(* Logix 5000 project; controller HP_SSC01hv vendor 1 type 14 code 158 rev 32.11; software revision 32.03; part 5 of 15 *)
(* tags used below, declared in another part *)
   A_C2_0300 : ALIAS FOR C2_FaultStandard.0;
   A_C2_0301 : ALIAS FOR C2_FaultStandard.1;
   A_C2_0302 : ALIAS FOR C2_FaultStandard.2;
   A_C2_0303 : ALIAS FOR C2_FaultStandard.3;
   A_C2_0305 : ALIAS FOR C2_FaultStandard.5;
   A_C2_0309 : ALIAS FOR C2_FaultStandard.9;
   A_C2_0310 : ALIAS FOR C2_FaultStandard.10;
   A_C2_0311 : ALIAS FOR C2_FaultStandard.11;
   A_C2_0312 : ALIAS FOR C2_FaultStandard.12;
   A_C2_0313 : ALIAS FOR C2_FaultStandard.13;
   A_C2_0314 : ALIAS FOR C2_FaultStandard.14;
   A_C2_0315 : ALIAS FOR C2_FaultStandard.15;
   A_C2_0317 : ALIAS FOR C2_FaultStandard.17;
   A_C2_0319 : ALIAS FOR C2_FaultStandard.19;
   A_C2_0321 : ALIAS FOR C2_FaultStandard.21;
   A_C2_0322 : ALIAS FOR C2_FaultStandard.22;
   A_C2_0323 : ALIAS FOR C2_FaultStandard.23;
   A_C2_0324 : ALIAS FOR C2_FaultStandard.24;
   A_C2_0325 : ALIAS FOR C2_FaultStandard.25;
   A_C2_0327 : ALIAS FOR C2_FaultStandard.27;
   A_C2_0328 : ALIAS FOR C2_FaultStandard.28;
   A_C2_0329 : ALIAS FOR C2_FaultStandard.29;
   A_C2_0330 : ALIAS FOR C2_FaultStandard.30;
   A_C2_0331 : ALIAS FOR C2_FaultStandard.31;
   A_C2_0404 : ALIAS FOR C2_Warning.4;
   A_C2_0406 : ALIAS FOR C2_Warning.6;
   A_C2_0407 : ALIAS FOR C2_Warning.7;
   A_C2_0408 : ALIAS FOR C2_Warning.8;
   A_C2_0409 : ALIAS FOR C2_Warning.9;
   A_C2_0412 : ALIAS FOR C2_Warning.12;
   A_C2_0413 : ALIAS FOR C2_Warning.13;
   A_C2_0414 : ALIAS FOR C2_Warning.14;
   A_C2_0415 : ALIAS FOR C2_Warning.15;
   A_C2_0416 : ALIAS FOR C2_Warning.16;
   A_C2_0424 : ALIAS FOR C2_Warning.24;
   A_C2_0427 : ALIAS FOR C2_Warning.27;
   A_C2_0428 : ALIAS FOR C2_Warning.28;
   A_C2_0430 : ALIAS FOR C2_Warning.30;
   C2_32HourTimers : TIMER[4];
   C2_All_DLY_OK : BOOL;
   C2_BrakeSequenceInProcess : BOOL;
   C2_BrakeTest : BOOL;
   C2_BrakeTestEndPosition : REAL;
   C2_BrakeTestFailed : BOOL;
   C2_BrakeTestLocalDisable : BOOL;
   C2_BrakeTestMAJ01 : MOTION_INSTRUCTION;
   C2_BrakeTestMessageNumber : DINT;
   C2_BrakeTestONS : BOOL;
   C2_BrakeTestSelected : BOOL;
   C2_BrakeTestSequence : DINT;
   C2_BrakeTestSequenceAlarms : DINT;
   C2_BrakeTestSequenceAlarmTimer : TIMER[16];
   C2_BrakeTestSequenceONS : DINT;
   C2_BrakeTestStartPosition : REAL;
   C2_BrakeTestStoppingDistance : REAL;
   C2_BrakeTestTimerHoldVel : TIMER;
   C2_BrakeTestWarning : BOOL;
   C2_DisableTimer : TIMER;
   C2_DumpTest : BOOL;
   C2_DumpValveFailedOff : BOOL;
   C2_DumpValveFailedOn : BOOL;
   C2_DumpValveMessageNumber : DINT;
   C2_DumpValveTestDelay : TIMER[4];
   C2_DumpValveTestDelay2 : TIMER;
   C2_DumpValveTestSelected : BOOL;
   C2_DumpValveTestSequence : DINT;
   C2_DumpValveTestSequenceAlarms : DINT;
   C2_DumpValveTestSequenceAlarmTimer : TIMER[8];
   C2_EncoderCounts : DINT;
   C2_EncoderCountsRaw : ALIAS FOR C2_RIO_AENT:3:I.PresentData;
   C2_EncoderDegree : REAL;
   C2_FaultDebounce : TIMER[16];
   C2_FaultHoldTimer : TIMER[4];
   C2_FaultHomeSwitchNotFound : BOOL;
   C2_FaultStandard : DINT;
   C2_HomeInputStatus : BOOL;
   C2_HomeSequence : DINT;
   C2_HomeSequenceAlarms : DINT;
   C2_HomeSwitchFaultK7KFailedOff : BOOL;
   C2_HomeSwitchFaultK7KFailedOn : BOOL;
   C2_HomeSwitchFaultSafeFailedOff : BOOL;
   C2_HomeSwitchFaultSafeFailedOn : BOOL;
   C2_IndexEnable : BOOL;
   C2_JogEnable : BOOL;
   C2_LIM_ALARM_B : ALIAS FOR C2_RIO_AENT:I.Data[1].0;
   C2_MaintEnable : BOOL;
   C2_MotorActualPositionX1000 : DINT;
   C2_MotorAverageVelocityX1000 : DINT;
   C2_MotorFan : ALIAS FOR C2_RIO_AENT:O.Data[2].0;
   C2_MSF : MOTION_INSTRUCTION;
   C2_MSO : MOTION_INSTRUCTION;
   C2_OIT_Current : DINT;
   C2_ONS_Fault : DINT;
   C2_RemoteBrakeAndHomeSequenceAlarms : DINT;
   C2_RemoteBrakeTestCMD : BOOL;
   C2_RemoteDumpTestCMD : BOOL;
   C2_ServoActionStatusOffDelay : TIMER;
   C2_ServoActionStatusOnDelay : TIMER;
   C2_ServoFanOverload : ALIAS FOR C2_RIO_AENT:I.Data[1].2;
   C2_SS_LocalRemote_1_IsRemote : ALIAS FOR C2_RIO_AENT:I.Data[1].3;
   C2_SS_RemoteMode : BOOL;
   C2_Warning : DINT;
   C2DumpValveTestSequenceONS : DINT;
   none : BOOL;
   RCS_CMD_RunInAuto : BOOL;
   RCS_SyncMotionEnable : BOOL;
   S_C2_EncoderPositionDegree : DINT;
   S_C2_ExecutePB : BOOL;
   S_C2_FaultReset : BOOL;
   S_C2_ModeLocal : BOOL;
   S_C2_ModeRemote : BOOL;
   S_C2_MotionEnabled : BOOL;
   S_C2_MSTOP_InputOK : BOOL;
   S_C2_NearOnPath : BOOL;
   S_C2_OffPath : BOOL;
   S_C2_OIT_FaultReset : BOOL;
   S_C2_OutputEnable : BOOL;
   S_C2_PressureOK : ALIAS FOR C2_Safe:I.Pt05Data;
   S_C2_SAFETY_ENABLE_1 : ALIAS FOR C2_Safe:O.Pt00Data;
   S_C2_SAFETY_ENABLE_2 : ALIAS FOR C2_Safe:O.Pt01Data;
   S_C2_Stop1_OK : BOOL;
   S_RCS_CMD_FaultReset : BOOL;
   STS_Enable_Rail : DINT;
   ZZZ_DIAG_A_C2_0302 : BOOL;
   ZZZ_DIAG_C2_AxisFault : DINT;
   ZZZ_DIAG_C2_AxisStatus : DINT;
   ZZZ_DIAG_C2_EnableRail : DINT;
   ZZZ_DIAG_C2_MotionStatus : DINT;
   ZZZ_DIAG_C2_MSF : MOTION_INSTRUCTION;
   ZZZ_DIAG_C2_MSO : MOTION_INSTRUCTION;
   ZZZ_DIAG_C2_OneTimeOnly : BOOL;
   ZZZ_DIAG_C2_OutputEnable : BOOL;
   ZZZ_DIAG_C2_OutputEnable_ACC : DINT;
   ZZZ_DIAG_ONS : DINT;
   ZZZ_DIAG_S_C2_OutputEnableTON : TIMER;
   ZZZ_DIAG_S_C2_SAFETY_ENABLE_1 : BOOL;
   ZZZ_DIAG_S_C2_SAFETY_ENABLE_2 : BOOL;

PROGRAM Carousel2   (* main routine C200_Main *)
VAR
   zzz_Test20 : BOOL;
   zzz_Test21 : BOOL;
END_VAR

ROUTINE C200_Main   (* ladder *)
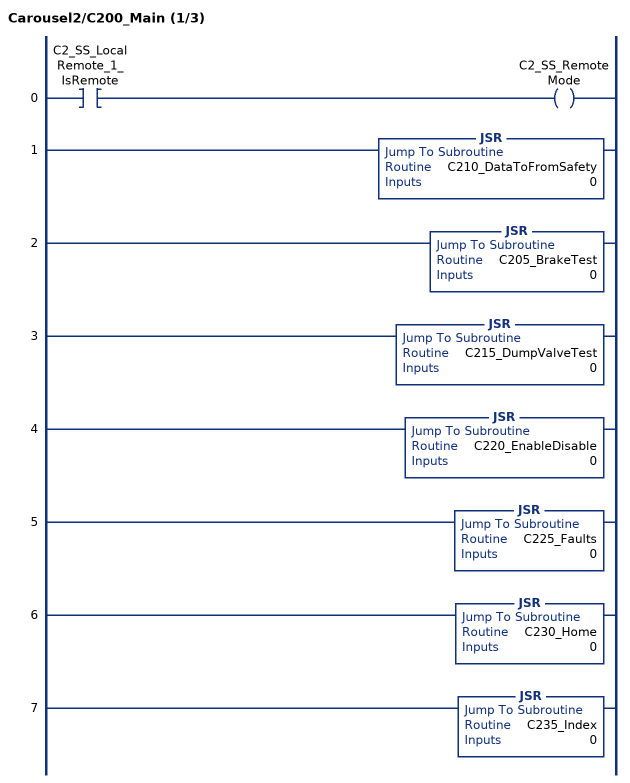
   0: XIC(C2_SS_LocalRemote_1_IsRemote)OTE(C2_SS_RemoteMode);
   1: JSR(C210_DataToFromSafety,0);
   2: JSR(C205_BrakeTest,0);
   3: JSR(C215_DumpValveTest,0);
   4: JSR(C220_EnableDisable,0);
   5: JSR(C225_Faults,0);
   6: JSR(C230_Home,0);
   7: JSR(C235_Index,0);
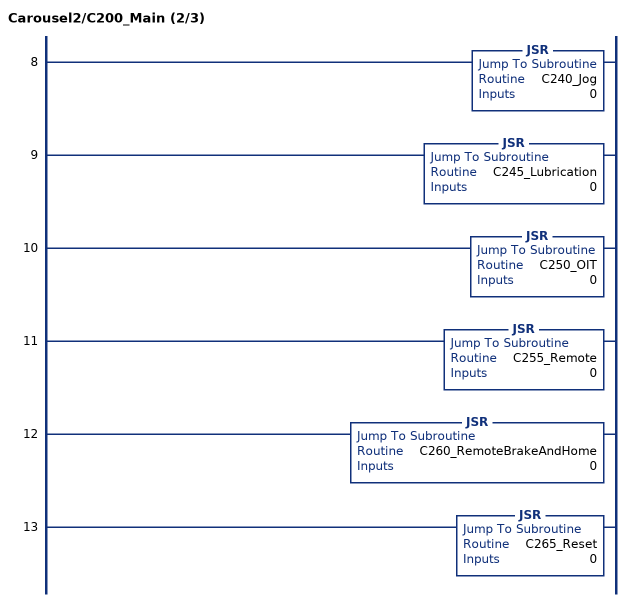
   8: JSR(C240_Jog,0);
   9: JSR(C245_Lubrication,0);
   10: JSR(C250_OIT,0);
   11: JSR(C255_Remote,0);
   12: JSR(C260_RemoteBrakeAndHome,0);
   13: JSR(C265_Reset,0);
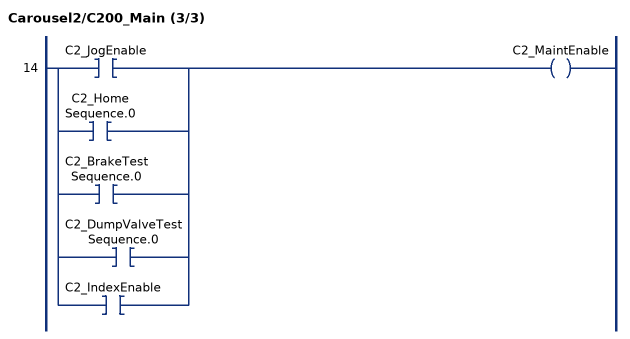
   14: [XIC(C2_JogEnable) ,XIC(C2_HomeSequence.0) ,XIC(C2_BrakeTestSequence.0) ,XIC(C2_DumpValveTestSequence.0) ,XIC(C2_IndexEnable) ]OTE(C2_MaintEnable);
END_ROUTINE

ROUTINE C205_BrakeTest   (* ladder *)
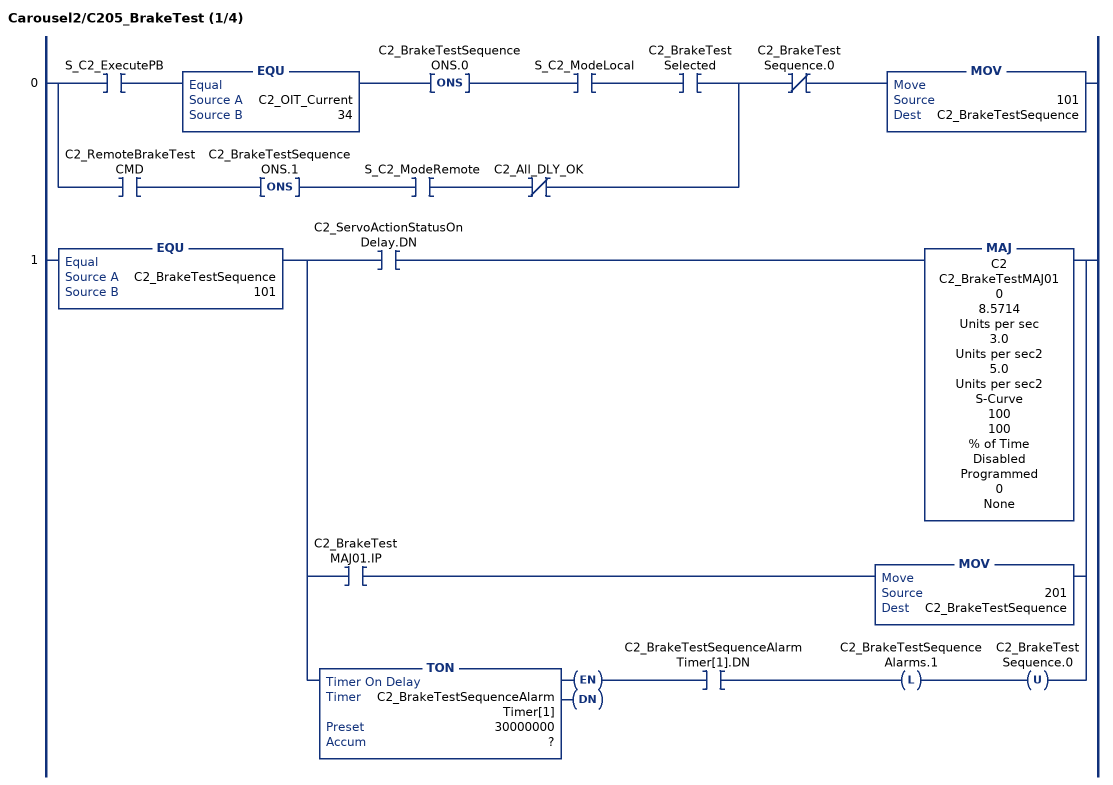
   0: [XIC(S_C2_ExecutePB) EQU(C2_OIT_Current,34) ONS(C2_BrakeTestSequenceONS.0) XIC(S_C2_ModeLocal) XIC(C2_BrakeTestSelected) ,XIC(C2_RemoteBrakeTestCMD) ONS(C2_BrakeTestSequenceONS.1) XIC(S_C2_ModeRemote) XIO(C2_All_DLY_OK) ]XIO(C2_BrakeTestSequence.0)MOV(101,C2_BrakeTestSequence);
   1: EQU(C2_BrakeTestSequence,101)[XIC(C2_ServoActionStatusOnDelay.DN) MAJ(C2,C2_BrakeTestMAJ01,0,8.5714,Units per sec,3.0,Units per sec2,5.0,Units per sec2,S-Curve,100,100,% of Time,Disabled,Programmed,0,None) ,XIC(C2_BrakeTestMAJ01.IP) MOV(201,C2_BrakeTestSequence) ,TON(C2_BrakeTestSequenceAlarmTimer[1],?,?) XIC(C2_BrakeTestSequenceAlarmTimer[1].DN) OTL(C2_BrakeTestSequenceAlarms.1) OTU(C2_BrakeTestSequence.0) ];
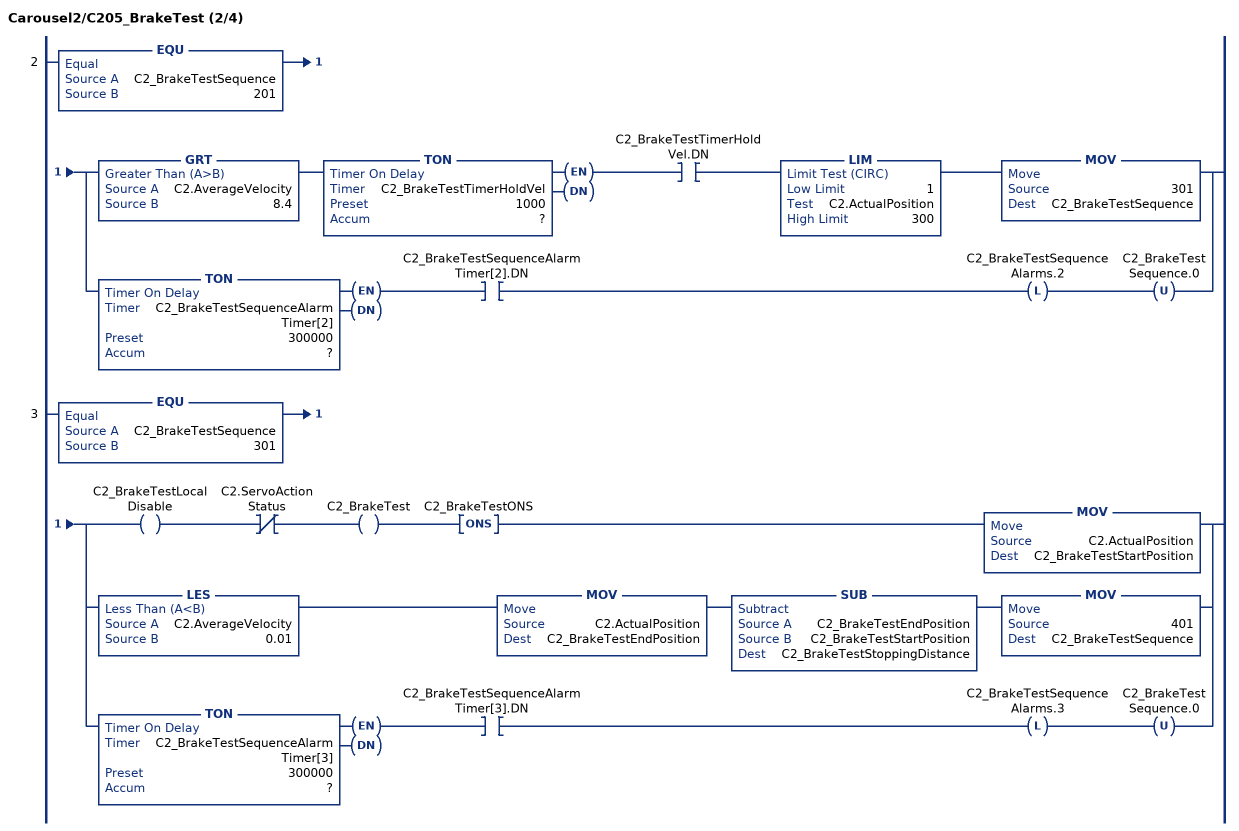
   2: EQU(C2_BrakeTestSequence,201)[GRT(C2.AverageVelocity,8.4) TON(C2_BrakeTestTimerHoldVel,?,?) XIC(C2_BrakeTestTimerHoldVel.DN) LIM(1,C2.ActualPosition,300) MOV(301,C2_BrakeTestSequence) ,TON(C2_BrakeTestSequenceAlarmTimer[2],?,?) XIC(C2_BrakeTestSequenceAlarmTimer[2].DN) OTL(C2_BrakeTestSequenceAlarms.2) OTU(C2_BrakeTestSequence.0) ];
   3: EQU(C2_BrakeTestSequence,301)[OTE(C2_BrakeTestLocalDisable) XIO(C2.ServoActionStatus) OTE(C2_BrakeTest) ONS(C2_BrakeTestONS) MOV(C2.ActualPosition,C2_BrakeTestStartPosition) ,LES(C2.AverageVelocity,0.01) MOV(C2.ActualPosition,C2_BrakeTestEndPosition) SUB(C2_BrakeTestEndPosition,C2_BrakeTestStartPosition,C2_BrakeTestStoppingDistance) MOV(401,C2_BrakeTestSequence) ,TON(C2_BrakeTestSequenceAlarmTimer[3],?,?) XIC(C2_BrakeTestSequenceAlarmTimer[3].DN) OTL(C2_BrakeTestSequenceAlarms.3) OTU(C2_BrakeTestSequence.0) ];
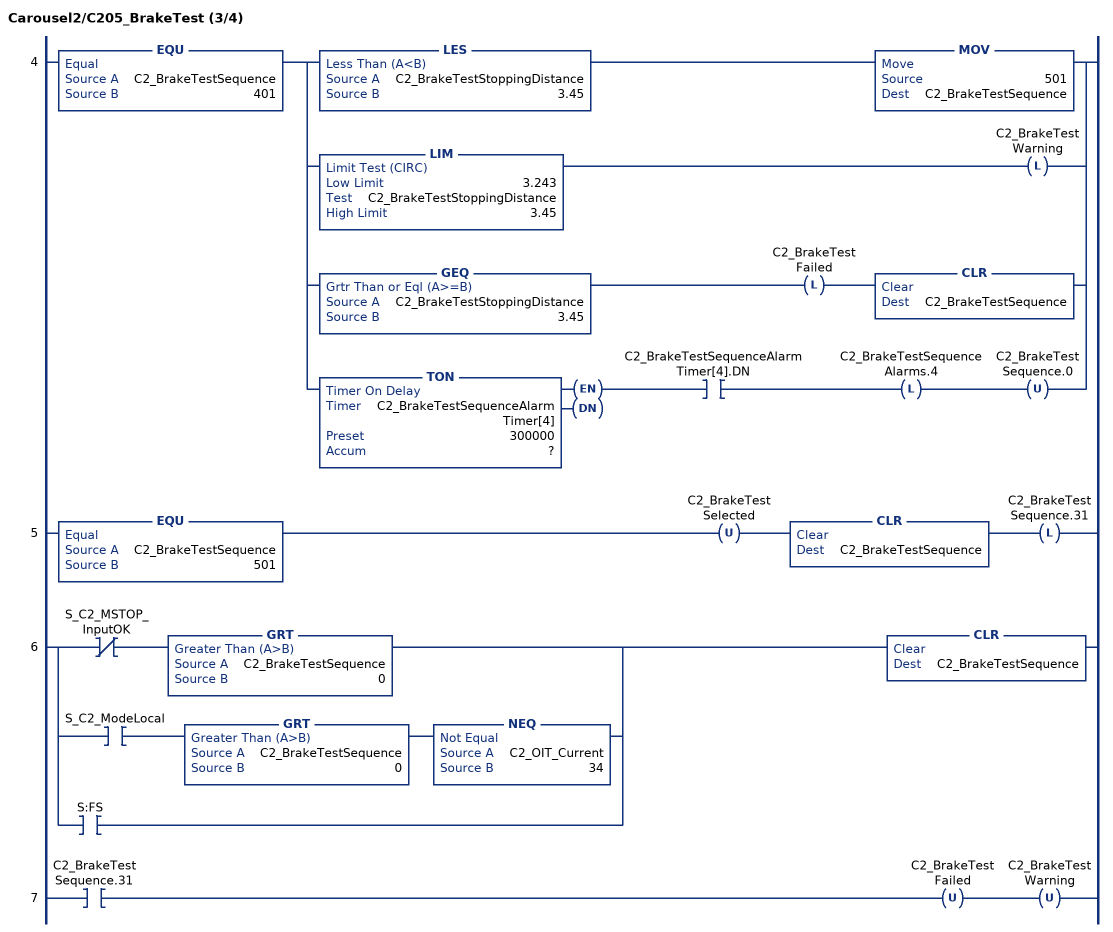
   4: EQU(C2_BrakeTestSequence,401)[LES(C2_BrakeTestStoppingDistance,3.45) MOV(501,C2_BrakeTestSequence) ,LIM(3.243,C2_BrakeTestStoppingDistance,3.45) OTL(C2_BrakeTestWarning) ,GEQ(C2_BrakeTestStoppingDistance,3.45) OTL(C2_BrakeTestFailed) CLR(C2_BrakeTestSequence) ,TON(C2_BrakeTestSequenceAlarmTimer[4],?,?) XIC(C2_BrakeTestSequenceAlarmTimer[4].DN) OTL(C2_BrakeTestSequenceAlarms.4) OTU(C2_BrakeTestSequence.0) ];
   5: EQU(C2_BrakeTestSequence,501)OTU(C2_BrakeTestSelected)CLR(C2_BrakeTestSequence)OTL(C2_BrakeTestSequence.31);
   6: [XIO(S_C2_MSTOP_InputOK) GRT(C2_BrakeTestSequence,0) ,XIC(S_C2_ModeLocal) GRT(C2_BrakeTestSequence,0) NEQ(C2_OIT_Current,34) ,XIC(S:FS) ]CLR(C2_BrakeTestSequence);
   7: XIC(C2_BrakeTestSequence.31)OTU(C2_BrakeTestFailed)OTU(C2_BrakeTestWarning);
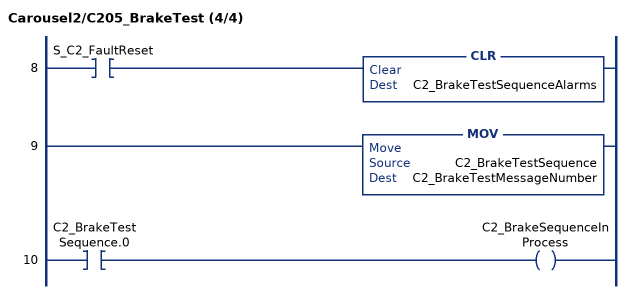
   8: XIC(S_C2_FaultReset)CLR(C2_BrakeTestSequenceAlarms);
   9: MOV(C2_BrakeTestSequence,C2_BrakeTestMessageNumber);
   10: XIC(C2_BrakeTestSequence.0)OTE(C2_BrakeSequenceInProcess);
END_ROUTINE

ROUTINE C210_DataToFromSafety   (* ladder *)
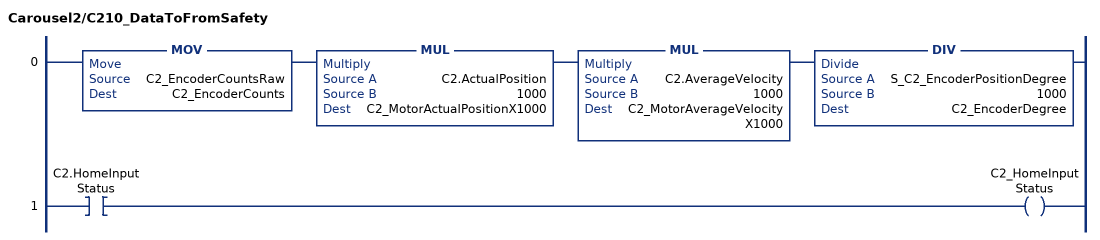
   0: MOV(C2_EncoderCountsRaw,C2_EncoderCounts)MUL(C2.ActualPosition,1000,C2_MotorActualPositionX1000)MUL(C2.AverageVelocity,1000,C2_MotorAverageVelocityX1000)DIV(S_C2_EncoderPositionDegree,1000,C2_EncoderDegree);
   1: XIC(C2.HomeInputStatus)OTE(C2_HomeInputStatus);
END_ROUTINE

ROUTINE C215_DumpValveTest   (* ladder *)
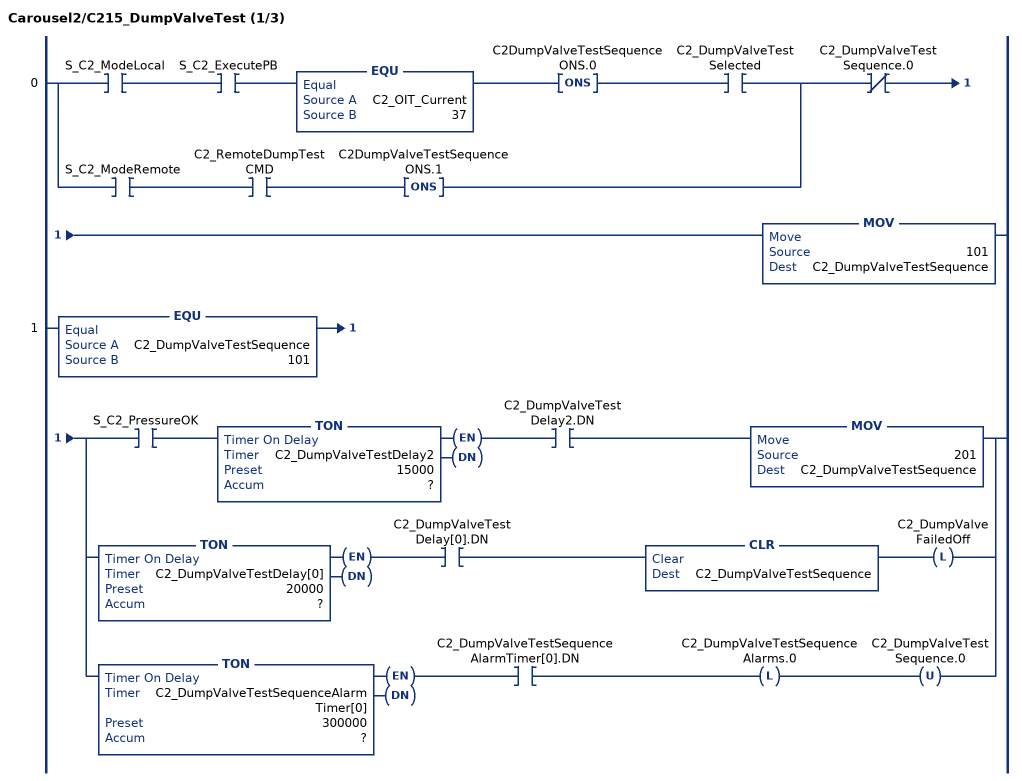
   0: [XIC(S_C2_ModeLocal) XIC(S_C2_ExecutePB) EQU(C2_OIT_Current,37) ONS(C2DumpValveTestSequenceONS.0) XIC(C2_DumpValveTestSelected) ,XIC(S_C2_ModeRemote) XIC(C2_RemoteDumpTestCMD) ONS(C2DumpValveTestSequenceONS.1) ]XIO(C2_DumpValveTestSequence.0)MOV(101,C2_DumpValveTestSequence);
   1: EQU(C2_DumpValveTestSequence,101)[XIC(S_C2_PressureOK) TON(C2_DumpValveTestDelay2,?,?) XIC(C2_DumpValveTestDelay2.DN) MOV(201,C2_DumpValveTestSequence) ,TON(C2_DumpValveTestDelay[0],?,?) XIC(C2_DumpValveTestDelay[0].DN) CLR(C2_DumpValveTestSequence) OTL(C2_DumpValveFailedOff) ,TON(C2_DumpValveTestSequenceAlarmTimer[0],?,?) XIC(C2_DumpValveTestSequenceAlarmTimer[0].DN) OTL(C2_DumpValveTestSequenceAlarms.0) OTU(C2_DumpValveTestSequence.0) ];
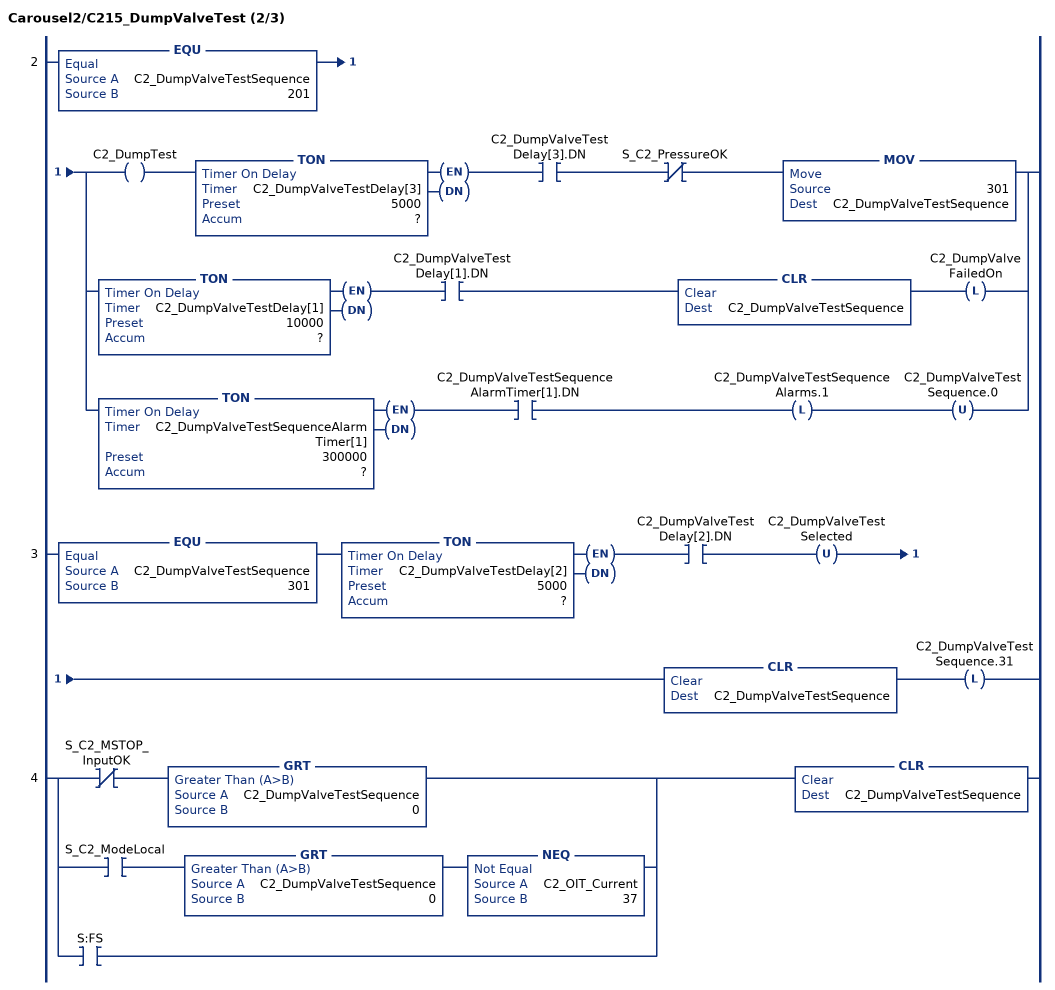
   2: EQU(C2_DumpValveTestSequence,201)[OTE(C2_DumpTest) TON(C2_DumpValveTestDelay[3],?,?) XIC(C2_DumpValveTestDelay[3].DN) XIO(S_C2_PressureOK) MOV(301,C2_DumpValveTestSequence) ,TON(C2_DumpValveTestDelay[1],?,?) XIC(C2_DumpValveTestDelay[1].DN) CLR(C2_DumpValveTestSequence) OTL(C2_DumpValveFailedOn) ,TON(C2_DumpValveTestSequenceAlarmTimer[1],?,?) XIC(C2_DumpValveTestSequenceAlarmTimer[1].DN) OTL(C2_DumpValveTestSequenceAlarms.1) OTU(C2_DumpValveTestSequence.0) ];
   3: EQU(C2_DumpValveTestSequence,301)TON(C2_DumpValveTestDelay[2],?,?)XIC(C2_DumpValveTestDelay[2].DN)OTU(C2_DumpValveTestSelected)CLR(C2_DumpValveTestSequence)OTL(C2_DumpValveTestSequence.31);
   4: [XIO(S_C2_MSTOP_InputOK) GRT(C2_DumpValveTestSequence,0) ,XIC(S_C2_ModeLocal) GRT(C2_DumpValveTestSequence,0) NEQ(C2_OIT_Current,37) ,XIC(S:FS) ]CLR(C2_DumpValveTestSequence);
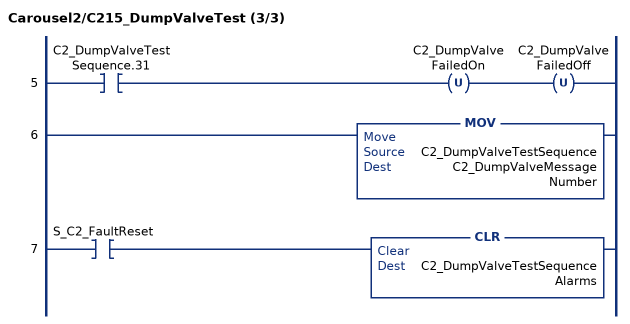
   5: XIC(C2_DumpValveTestSequence.31)OTU(C2_DumpValveFailedOn)OTU(C2_DumpValveFailedOff);
   6: MOV(C2_DumpValveTestSequence,C2_DumpValveMessageNumber);
   7: XIC(S_C2_FaultReset)CLR(C2_DumpValveTestSequenceAlarms);
END_ROUTINE

ROUTINE C220_EnableDisable   (* ladder *)
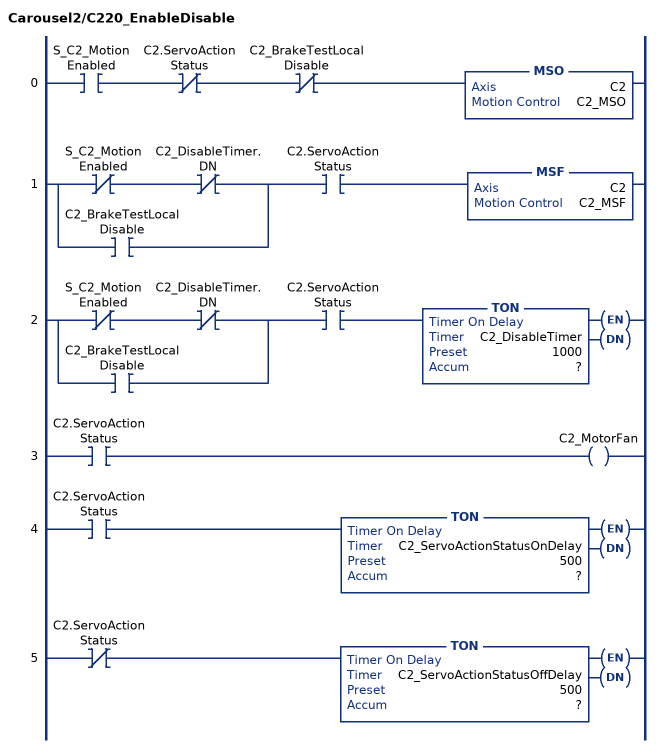
   0: XIC(S_C2_MotionEnabled)XIO(C2.ServoActionStatus)XIO(C2_BrakeTestLocalDisable)MSO(C2,C2_MSO);
   1: [XIO(S_C2_MotionEnabled) XIO(C2_DisableTimer.DN) ,XIC(C2_BrakeTestLocalDisable) ]XIC(C2.ServoActionStatus)MSF(C2,C2_MSF);
   2: [XIO(S_C2_MotionEnabled) XIO(C2_DisableTimer.DN) ,XIC(C2_BrakeTestLocalDisable) ]XIC(C2.ServoActionStatus)TON(C2_DisableTimer,?,?);
   3: XIC(C2.ServoActionStatus)OTE(C2_MotorFan);
   4: XIC(C2.ServoActionStatus)TON(C2_ServoActionStatusOnDelay,?,?);
   5: XIO(C2.ServoActionStatus)TON(C2_ServoActionStatusOffDelay,?,?);
END_ROUTINE

ROUTINE C225_Faults   (* ladder *)
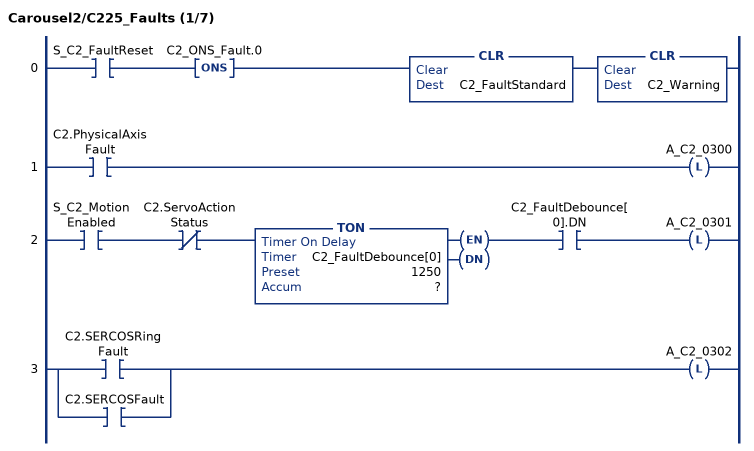
   0: XIC(S_C2_FaultReset)ONS(C2_ONS_Fault.0)CLR(C2_FaultStandard)CLR(C2_Warning);
   1: XIC(C2.PhysicalAxisFault)OTL(A_C2_0300);
   2: XIC(S_C2_MotionEnabled)XIO(C2.ServoActionStatus)TON(C2_FaultDebounce[0],?,?)XIC(C2_FaultDebounce[0].DN)OTL(A_C2_0301);
   3: [XIC(C2.SERCOSRingFault) ,XIC(C2.SERCOSFault) ]OTL(A_C2_0302);
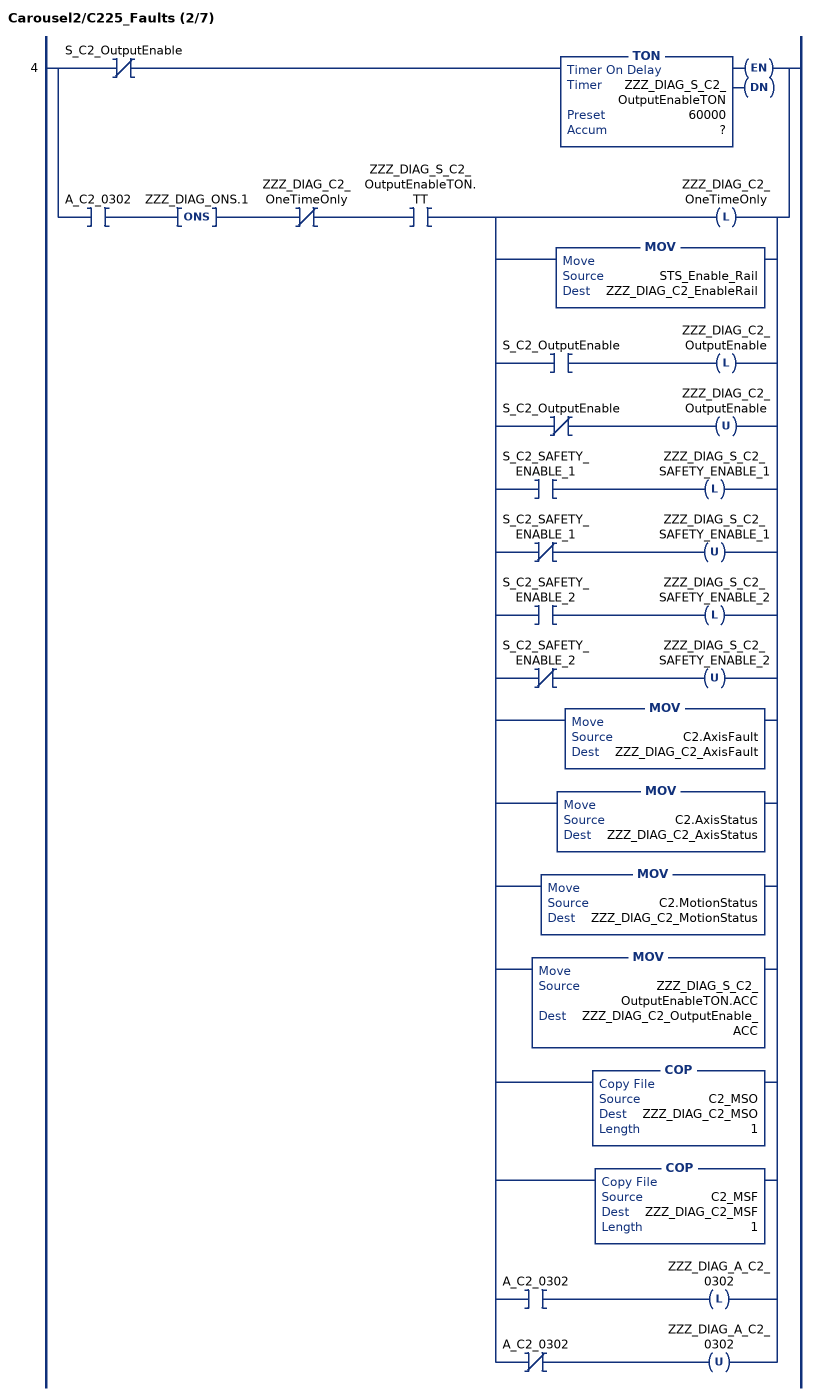
   4: [XIO(S_C2_OutputEnable) TON(ZZZ_DIAG_S_C2_OutputEnableTON,?,?) ,XIC(A_C2_0302) ONS(ZZZ_DIAG_ONS.1) XIO(ZZZ_DIAG_C2_OneTimeOnly) XIC(ZZZ_DIAG_S_C2_OutputEnableTON.TT) [OTL(ZZZ_DIAG_C2_OneTimeOnly) ,MOV(STS_Enable_Rail,ZZZ_DIAG_C2_EnableRail) ,XIC(S_C2_OutputEnable) OTL(ZZZ_DIAG_C2_OutputEnable) ,XIO(S_C2_OutputEnable) OTU(ZZZ_DIAG_C2_OutputEnable) ,XIC(S_C2_SAFETY_ENABLE_1) OTL(ZZZ_DIAG_S_C2_SAFETY_ENABLE_1) ,XIO(S_C2_SAFETY_ENABLE_1) OTU(ZZZ_DIAG_S_C2_SAFETY_ENABLE_1) ,XIC(S_C2_SAFETY_ENABLE_2) OTL(ZZZ_DIAG_S_C2_SAFETY_ENABLE_2) ,XIO(S_C2_SAFETY_ENABLE_2) OTU(ZZZ_DIAG_S_C2_SAFETY_ENABLE_2) ,MOV(C2.AxisFault,ZZZ_DIAG_C2_AxisFault) ,MOV(C2.AxisStatus,ZZZ_DIAG_C2_AxisStatus) ,MOV(C2.MotionStatus,ZZZ_DIAG_C2_MotionStatus) ,MOV(ZZZ_DIAG_S_C2_OutputEnableTON.ACC,ZZZ_DIAG_C2_OutputEnable_ACC) ,COP(C2_MSO,ZZZ_DIAG_C2_MSO,1) ,COP(C2_MSF,ZZZ_DIAG_C2_MSF,1) ,XIC(A_C2_0302) OTL(ZZZ_DIAG_A_C2_0302) ,XIO(A_C2_0302) OTU(ZZZ_DIAG_A_C2_0302) ] ];
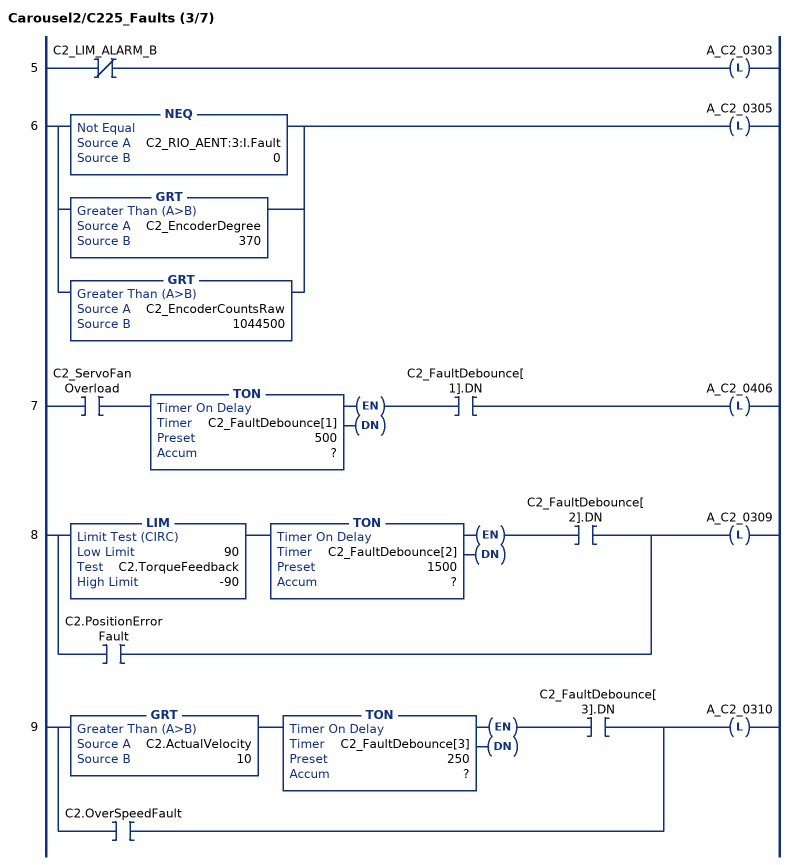
   5: XIO(C2_LIM_ALARM_B)OTL(A_C2_0303);
   6: [NEQ(C2_RIO_AENT:3:I.Fault,0) ,GRT(C2_EncoderDegree,370) ,GRT(C2_EncoderCountsRaw,1044500) ]OTL(A_C2_0305);
   7: XIC(C2_ServoFanOverload)TON(C2_FaultDebounce[1],?,?)XIC(C2_FaultDebounce[1].DN)OTL(A_C2_0406);
   8: [LIM(90,C2.TorqueFeedback,-90) TON(C2_FaultDebounce[2],?,?) XIC(C2_FaultDebounce[2].DN) ,XIC(C2.PositionErrorFault) ]OTL(A_C2_0309);
   9: [GRT(C2.ActualVelocity,10) TON(C2_FaultDebounce[3],?,?) XIC(C2_FaultDebounce[3].DN) ,XIC(C2.OverSpeedFault) ]OTL(A_C2_0310);
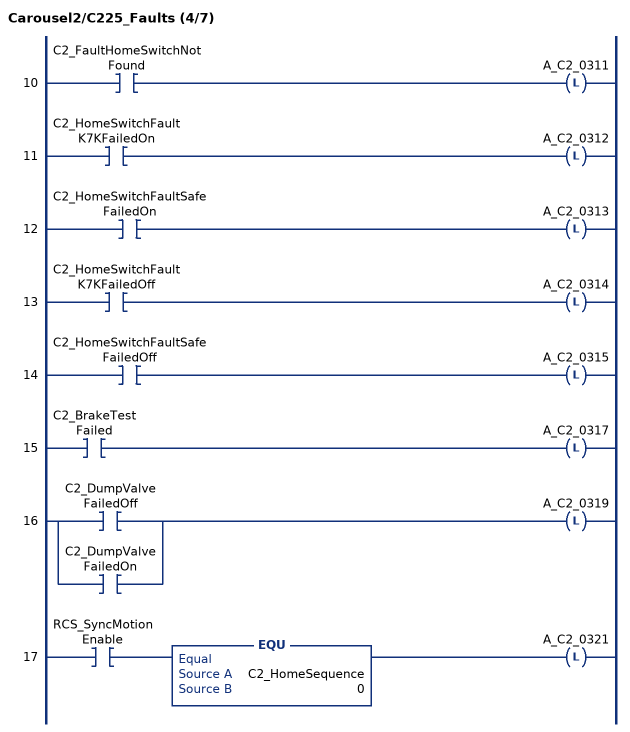
   10: XIC(C2_FaultHomeSwitchNotFound)OTL(A_C2_0311);
   11: XIC(C2_HomeSwitchFaultK7KFailedOn)OTL(A_C2_0312);
   12: XIC(C2_HomeSwitchFaultSafeFailedOn)OTL(A_C2_0313);
   13: XIC(C2_HomeSwitchFaultK7KFailedOff)OTL(A_C2_0314);
   14: XIC(C2_HomeSwitchFaultSafeFailedOff)OTL(A_C2_0315);
   15: XIC(C2_BrakeTestFailed)OTL(A_C2_0317);
   16: [XIC(C2_DumpValveFailedOff) ,XIC(C2_DumpValveFailedOn) ]OTL(A_C2_0319);
   17: XIC(RCS_SyncMotionEnable)EQU(C2_HomeSequence,0)OTL(A_C2_0321);
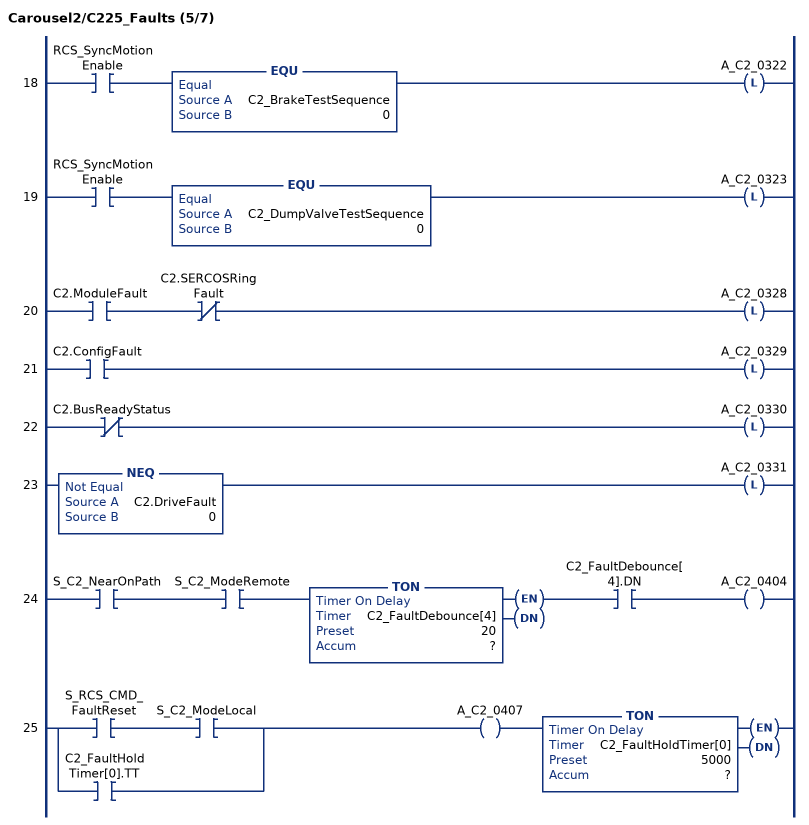
   18: XIC(RCS_SyncMotionEnable)EQU(C2_BrakeTestSequence,0)OTL(A_C2_0322);
   19: XIC(RCS_SyncMotionEnable)EQU(C2_DumpValveTestSequence,0)OTL(A_C2_0323);
   20: XIC(C2.ModuleFault)XIO(C2.SERCOSRingFault)OTL(A_C2_0328);
   21: XIC(C2.ConfigFault)OTL(A_C2_0329);
   22: XIO(C2.BusReadyStatus)OTL(A_C2_0330);
   23: NEQ(C2.DriveFault,0)OTL(A_C2_0331);
   24: XIC(S_C2_NearOnPath)XIC(S_C2_ModeRemote)TON(C2_FaultDebounce[4],?,?)XIC(C2_FaultDebounce[4].DN)OTE(A_C2_0404);
   25: [XIC(S_RCS_CMD_FaultReset) XIC(S_C2_ModeLocal) ,XIC(C2_FaultHoldTimer[0].TT) ]OTE(A_C2_0407)TON(C2_FaultHoldTimer[0],?,?);
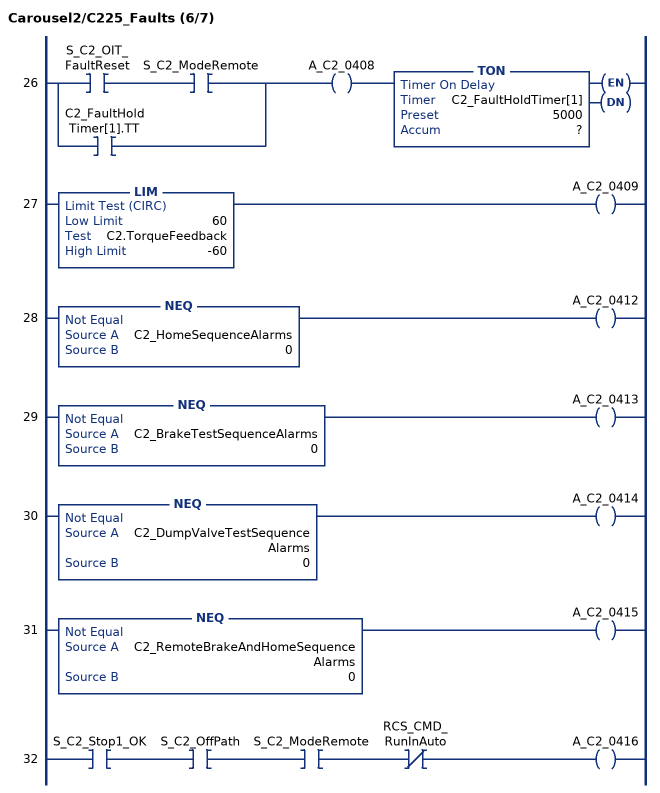
   26: [XIC(S_C2_OIT_FaultReset) XIC(S_C2_ModeRemote) ,XIC(C2_FaultHoldTimer[1].TT) ]OTE(A_C2_0408)TON(C2_FaultHoldTimer[1],?,?);
   27: LIM(60,C2.TorqueFeedback,-60)OTE(A_C2_0409);
   28: NEQ(C2_HomeSequenceAlarms,0)OTE(A_C2_0412);
   29: NEQ(C2_BrakeTestSequenceAlarms,0)OTE(A_C2_0413);
   30: NEQ(C2_DumpValveTestSequenceAlarms,0)OTE(A_C2_0414);
   31: NEQ(C2_RemoteBrakeAndHomeSequenceAlarms,0)OTE(A_C2_0415);
   32: XIC(S_C2_Stop1_OK)XIC(S_C2_OffPath)XIC(S_C2_ModeRemote)XIO(RCS_CMD_RunInAuto)OTE(A_C2_0416);
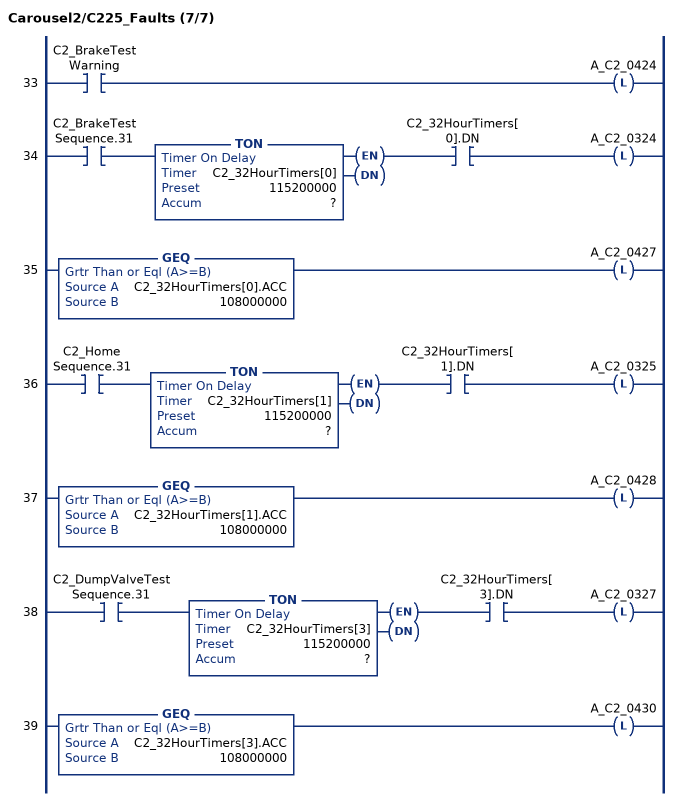
   33: XIC(C2_BrakeTestWarning)OTL(A_C2_0424);
   34: XIC(C2_BrakeTestSequence.31)TON(C2_32HourTimers[0],?,?)XIC(C2_32HourTimers[0].DN)OTL(A_C2_0324);
   35: GEQ(C2_32HourTimers[0].ACC,108000000)OTL(A_C2_0427);
   36: XIC(C2_HomeSequence.31)TON(C2_32HourTimers[1],?,?)XIC(C2_32HourTimers[1].DN)OTL(A_C2_0325);
   37: GEQ(C2_32HourTimers[1].ACC,108000000)OTL(A_C2_0428);
   38: XIC(C2_DumpValveTestSequence.31)TON(C2_32HourTimers[3],?,?)XIC(C2_32HourTimers[3].DN)OTL(A_C2_0327);
   39: GEQ(C2_32HourTimers[3].ACC,108000000)OTL(A_C2_0430);
END_ROUTINE
